{attribute 'qualified_only'}
{attribute 'strict'}
TYPE E_SafetyCtrlState :
(
	enum_member := 0
);
END_TYPE

(* stored: Version 1.1.0.1, ProductVersion 3.1.4024.9
   DUT E_SafetyCtrlState: Id {b55b7e1b-4ed8-4673-adbc-aff2998116f9} *)
